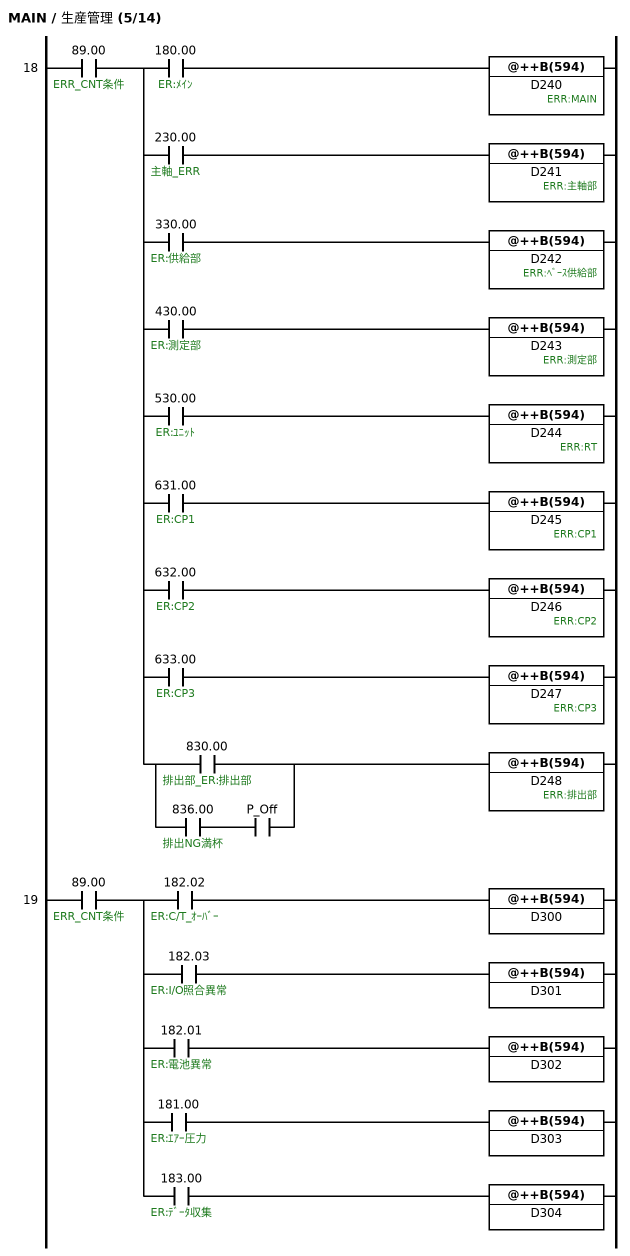
; [picture p24: MAIN / 生産管理, rungs 18-19]
; rung 18
LD 89.00  ; ERR_CNT条件
OUT TR0
AND 180.00  ; ER:ﾒｲﾝ
@++B(594) D240  ; ERR:MAIN
LD TR0
AND 230.00  ; 主軸_ERR
@++B(594) D241  ; ERR:主軸部
LD TR0
AND 330.00  ; ER:供給部
@++B(594) D242  ; ERR:ﾍﾞｰｽ供給部
LD TR0
AND 430.00  ; ER:測定部
@++B(594) D243  ; ERR:測定部
LD TR0
AND 530.00  ; ER:ﾕﾆｯﾄ
@++B(594) D244  ; ERR:RT
LD TR0
AND 631.00  ; ER:CP1
@++B(594) D245  ; ERR:CP1
LD TR0
AND 632.00  ; ER:CP2
@++B(594) D246  ; ERR:CP2
LD TR0
AND 633.00  ; ER:CP3
@++B(594) D247  ; ERR:CP3
LD TR0
LD 830.00  ; 排出部_ER:排出部
LD 836.00  ; 排出NG満杯
AND P_Off
ORLD
ANDLD
@++B(594) D248  ; ERR:排出部
; rung 19
LD 89.00  ; ERR_CNT条件
OUT TR0
AND 182.02  ; ER:C/T_ｵｰﾊﾞｰ
@++B(594) D300
LD TR0
AND 182.03  ; ER:I/O照合異常
@++B(594) D301
LD TR0
AND 182.01  ; ER:電池異常
@++B(594) D302
LD TR0
AND 181.00  ; ER:ｴｱｰ圧力
@++B(594) D303
LD TR0
AND 183.00  ; ER:ﾃﾞｰﾀ収集
@++B(594) D304

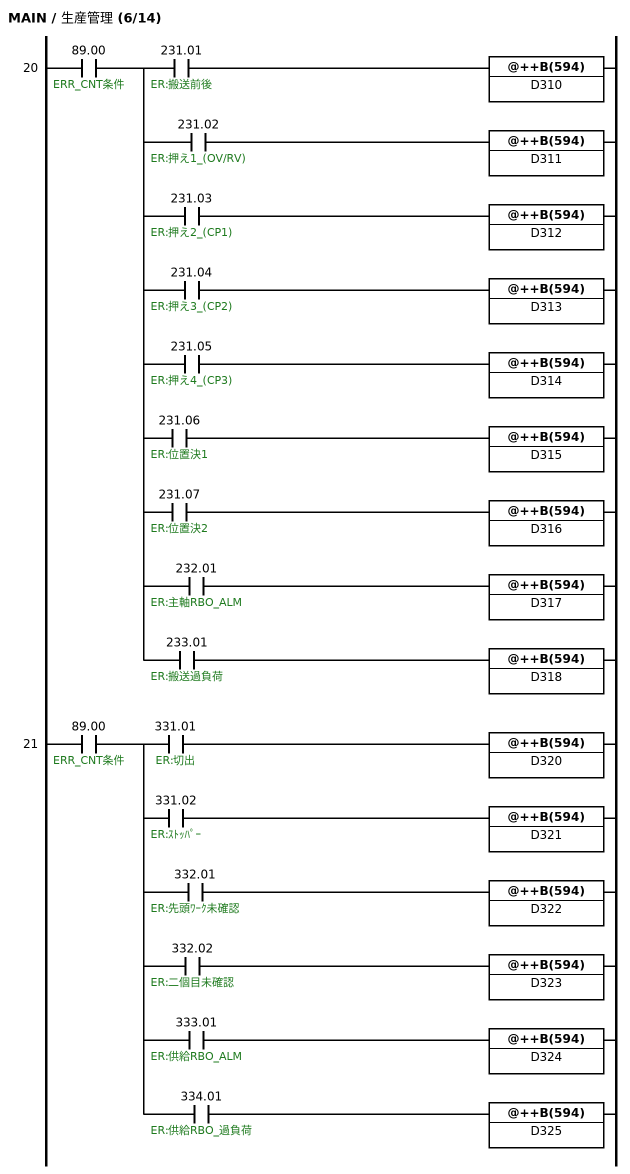
; rung 20
LD 89.00  ; ERR_CNT条件
OUT TR0
AND 231.01  ; ER:搬送前後
@++B(594) D310
LD TR0
AND 231.02  ; ER:押え1_(OV/RV)
@++B(594) D311
LD TR0
AND 231.03  ; ER:押え2_(CP1)
@++B(594) D312
LD TR0
AND 231.04  ; ER:押え3_(CP2)
@++B(594) D313
LD TR0
AND 231.05  ; ER:押え4_(CP3)
@++B(594) D314
LD TR0
AND 231.06  ; ER:位置決1
@++B(594) D315
LD TR0
AND 231.07  ; ER:位置決2
@++B(594) D316
LD TR0
AND 232.01  ; ER:主軸RBO_ALM
@++B(594) D317
LD TR0
AND 233.01  ; ER:搬送過負荷
@++B(594) D318
; rung 21
LD 89.00  ; ERR_CNT条件
OUT TR0
AND 331.01  ; ER:切出
@++B(594) D320
LD TR0
AND 331.02  ; ER:ｽﾄｯﾊﾟｰ
@++B(594) D321
LD TR0
AND 332.01  ; ER:先頭ﾜｰｸ未確認
@++B(594) D322
LD TR0
AND 332.02  ; ER:二個目未確認
@++B(594) D323
LD TR0
AND 333.01  ; ER:供給RBO_ALM
@++B(594) D324
LD TR0
AND 334.01  ; ER:供給RBO_過負荷
@++B(594) D325

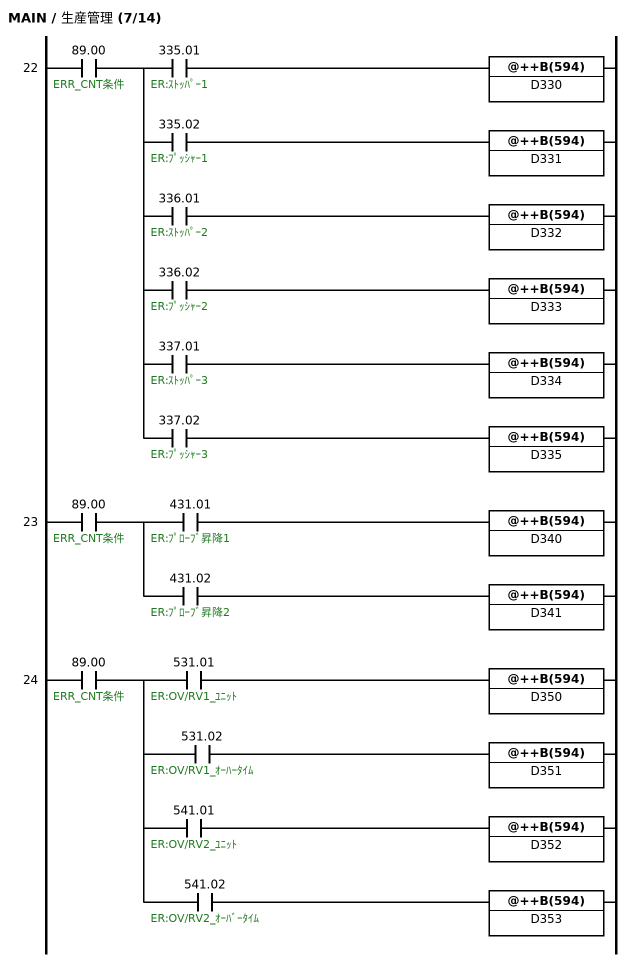
; rung 22
LD 89.00  ; ERR_CNT条件
OUT TR0
AND 335.01  ; ER:ｽﾄｯﾊﾟｰ1
@++B(594) D330
LD TR0
AND 335.02  ; ER:ﾌﾟｯｼｬｰ1
@++B(594) D331
LD TR0
AND 336.01  ; ER:ｽﾄｯﾊﾟｰ2
@++B(594) D332
LD TR0
AND 336.02  ; ER:ﾌﾟｯｼｬｰ2
@++B(594) D333
LD TR0
AND 337.01  ; ER:ｽﾄｯﾊﾟｰ3
@++B(594) D334
LD TR0
AND 337.02  ; ER:ﾌﾟｯｼｬｰ3
@++B(594) D335
; rung 23
LD 89.00  ; ERR_CNT条件
OUT TR0
AND 431.01  ; ER:ﾌﾟﾛｰﾌﾞ昇降1
@++B(594) D340
LD TR0
AND 431.02  ; ER:ﾌﾟﾛｰﾌﾞ昇降2
@++B(594) D341
; rung 24
LD 89.00  ; ERR_CNT条件
OUT TR0
AND 531.01  ; ER:OV/RV1_ﾕﾆｯﾄ
@++B(594) D350
LD TR0
AND 531.02  ; ER:OV/RV1_ｵｰﾊｰﾀｲﾑ
@++B(594) D351
LD TR0
AND 541.01  ; ER:OV/RV2_ﾕﾆｯﾄ
@++B(594) D352
LD TR0
AND 541.02  ; ER:OV/RV2_ｵｰﾊﾞｰﾀｲﾑ
@++B(594) D353

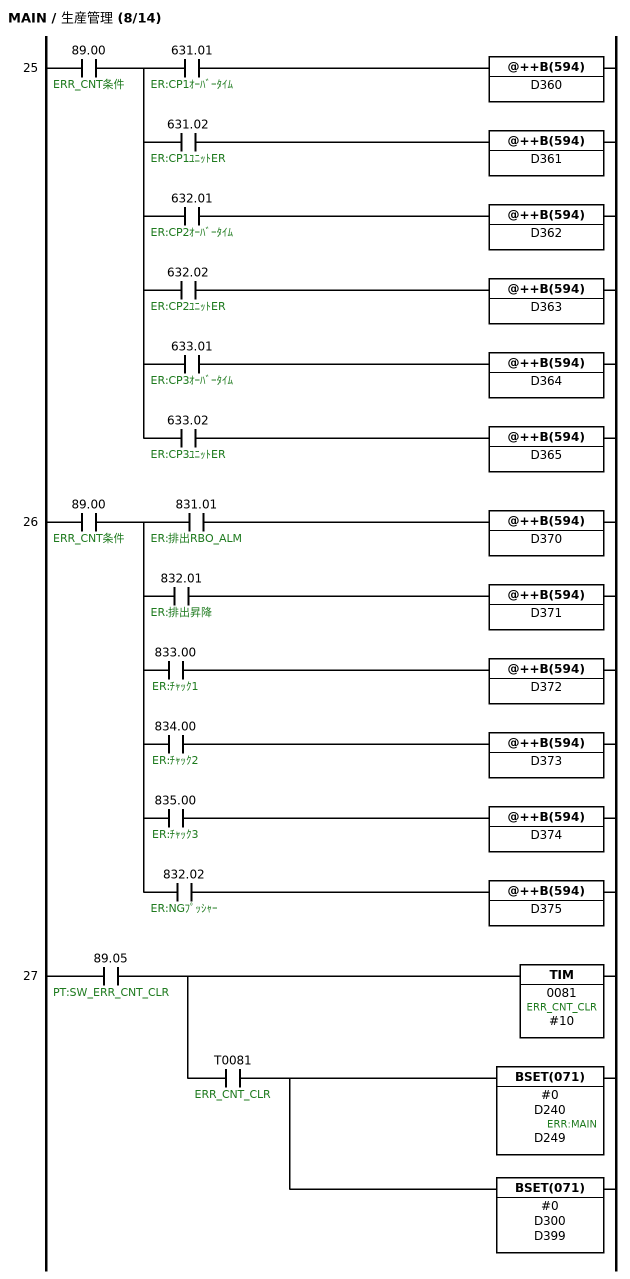
; rung 25
LD 89.00  ; ERR_CNT条件
OUT TR0
AND 631.01  ; ER:CP1ｵｰﾊﾞｰﾀｲﾑ
@++B(594) D360
LD TR0
AND 631.02  ; ER:CP1ﾕﾆｯﾄER
@++B(594) D361
LD TR0
AND 632.01  ; ER:CP2ｵｰﾊﾞｰﾀｲﾑ
@++B(594) D362
LD TR0
AND 632.02  ; ER:CP2ﾕﾆｯﾄER
@++B(594) D363
LD TR0
AND 633.01  ; ER:CP3ｵｰﾊﾞｰﾀｲﾑ
@++B(594) D364
LD TR0
AND 633.02  ; ER:CP3ﾕﾆｯﾄER
@++B(594) D365
; rung 26
LD 89.00  ; ERR_CNT条件
OUT TR0
AND 831.01  ; ER:排出RBO_ALM
@++B(594) D370
LD TR0
AND 832.01  ; ER:排出昇降
@++B(594) D371
LD TR0
AND 833.00  ; ER:ﾁｬｯｸ1
@++B(594) D372
LD TR0
AND 834.00  ; ER:ﾁｬｯｸ2
@++B(594) D373
LD TR0
AND 835.00  ; ER:ﾁｬｯｸ3
@++B(594) D374
LD TR0
AND 832.02  ; ER:NGﾌﾟｯｼｬｰ
@++B(594) D375
; rung 27
LD 89.05  ; PT:SW_ERR_CNT_CLR
TIM 0081 #10  ; ERR_CNT_CLR
AND T0081  ; ERR_CNT_CLR
BSET(071) #0 D240 D249  ; ERR:MAIN
BSET(071) #0 D300 D399

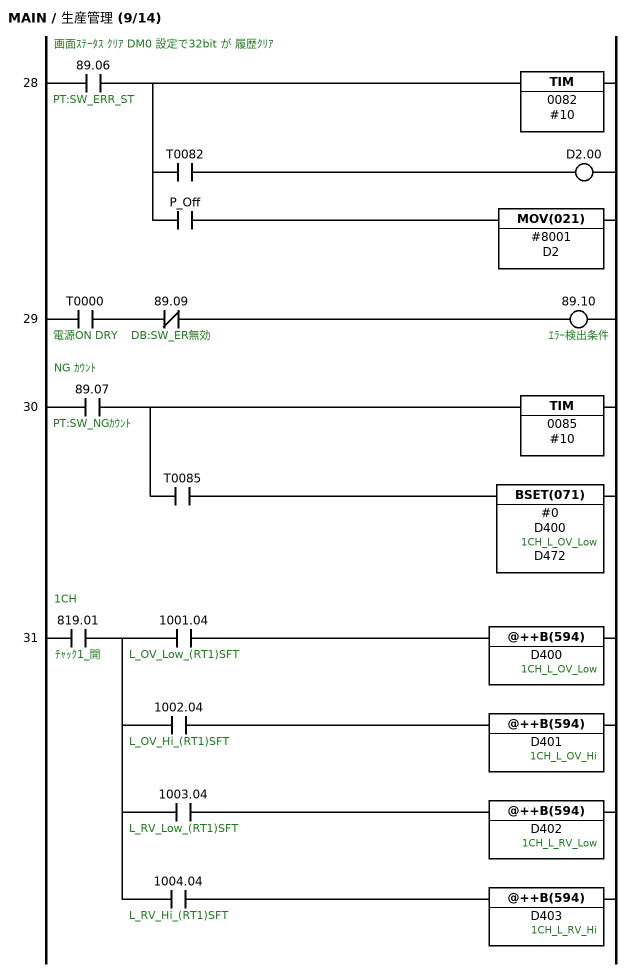
; rung 28: 画面ｽﾃｰﾀｽ ｸﾘｱ DM0 設定で32bit が 履歴ｸﾘｱ
LD 89.06  ; PT:SW_ERR_ST
OUT TR0
TIM 0082 #10
AND T0082
OUT D2.00
LD TR0
AND P_Off
MOV(021) #8001 D2
; rung 29
LD T0000  ; 電源ON DRY
ANDNOT 89.09  ; DB:SW_ER無効
OUT 89.10  ; ｴﾗｰ検出条件
; rung 30: NG ｶｳﾝﾄ
LD 89.07  ; PT:SW_NGｶｳﾝﾄ
TIM 0085 #10
AND T0085
BSET(071) #0 D400 D472  ; 1CH_L_OV_Low
; rung 31: 1CH
LD 819.01  ; ﾁｬｯｸ1_開
OUT TR0
AND 1001.04  ; L_OV_Low_(RT1)SFT
@++B(594) D400  ; 1CH_L_OV_Low
LD TR0
AND 1002.04  ; L_OV_Hi_(RT1)SFT
@++B(594) D401  ; 1CH_L_OV_Hi
LD TR0
AND 1003.04  ; L_RV_Low_(RT1)SFT
@++B(594) D402  ; 1CH_L_RV_Low
LD TR0
AND 1004.04  ; L_RV_Hi_(RT1)SFT
@++B(594) D403  ; 1CH_L_RV_Hi

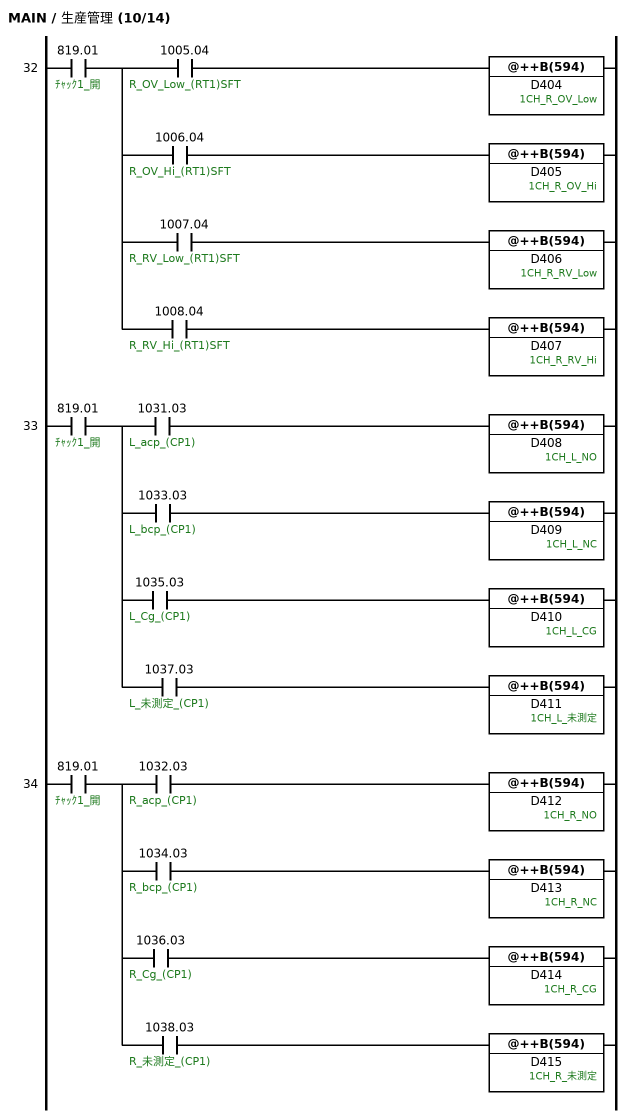
; rung 32
LD 819.01  ; ﾁｬｯｸ1_開
OUT TR0
AND 1005.04  ; R_OV_Low_(RT1)SFT
@++B(594) D404  ; 1CH_R_OV_Low
LD TR0
AND 1006.04  ; R_OV_Hi_(RT1)SFT
@++B(594) D405  ; 1CH_R_OV_Hi
LD TR0
AND 1007.04  ; R_RV_Low_(RT1)SFT
@++B(594) D406  ; 1CH_R_RV_Low
LD TR0
AND 1008.04  ; R_RV_Hi_(RT1)SFT
@++B(594) D407  ; 1CH_R_RV_Hi
; rung 33
LD 819.01  ; ﾁｬｯｸ1_開
OUT TR0
AND 1031.03  ; L_acp_(CP1)
@++B(594) D408  ; 1CH_L_NO
LD TR0
AND 1033.03  ; L_bcp_(CP1)
@++B(594) D409  ; 1CH_L_NC
LD TR0
AND 1035.03  ; L_Cg_(CP1)
@++B(594) D410  ; 1CH_L_CG
LD TR0
AND 1037.03  ; L_未測定_(CP1)
@++B(594) D411  ; 1CH_L_未測定
; rung 34
LD 819.01  ; ﾁｬｯｸ1_開
OUT TR0
AND 1032.03  ; R_acp_(CP1)
@++B(594) D412  ; 1CH_R_NO
LD TR0
AND 1034.03  ; R_bcp_(CP1)
@++B(594) D413  ; 1CH_R_NC
LD TR0
AND 1036.03  ; R_Cg_(CP1)
@++B(594) D414  ; 1CH_R_CG
LD TR0
AND 1038.03  ; R_未測定_(CP1)
@++B(594) D415  ; 1CH_R_未測定

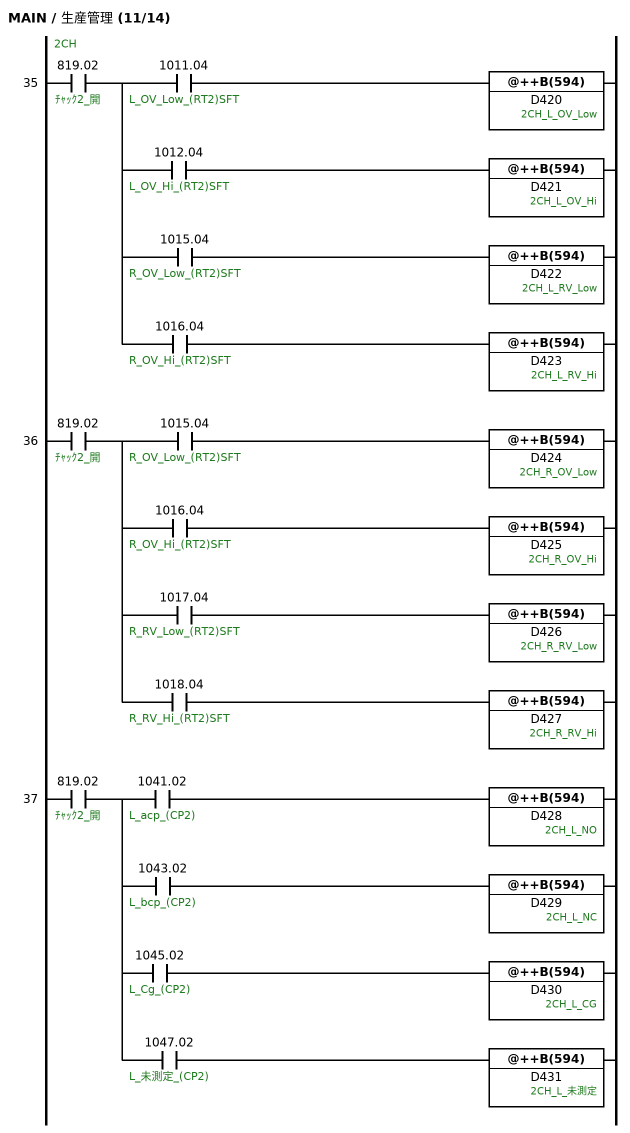
; rung 35: 2CH
LD 819.02  ; ﾁｬｯｸ2_開
OUT TR0
AND 1011.04  ; L_OV_Low_(RT2)SFT
@++B(594) D420  ; 2CH_L_OV_Low
LD TR0
AND 1012.04  ; L_OV_Hi_(RT2)SFT
@++B(594) D421  ; 2CH_L_OV_Hi
LD TR0
AND 1015.04  ; R_OV_Low_(RT2)SFT
@++B(594) D422  ; 2CH_L_RV_Low
LD TR0
AND 1016.04  ; R_OV_Hi_(RT2)SFT
@++B(594) D423  ; 2CH_L_RV_Hi
; rung 36
LD 819.02  ; ﾁｬｯｸ2_開
OUT TR0
AND 1015.04  ; R_OV_Low_(RT2)SFT
@++B(594) D424  ; 2CH_R_OV_Low
LD TR0
AND 1016.04  ; R_OV_Hi_(RT2)SFT
@++B(594) D425  ; 2CH_R_OV_Hi
LD TR0
AND 1017.04  ; R_RV_Low_(RT2)SFT
@++B(594) D426  ; 2CH_R_RV_Low
LD TR0
AND 1018.04  ; R_RV_Hi_(RT2)SFT
@++B(594) D427  ; 2CH_R_RV_Hi
; rung 37
LD 819.02  ; ﾁｬｯｸ2_開
OUT TR0
AND 1041.02  ; L_acp_(CP2)
@++B(594) D428  ; 2CH_L_NO
LD TR0
AND 1043.02  ; L_bcp_(CP2)
@++B(594) D429  ; 2CH_L_NC
LD TR0
AND 1045.02  ; L_Cg_(CP2)
@++B(594) D430  ; 2CH_L_CG
LD TR0
AND 1047.02  ; L_未測定_(CP2)
@++B(594) D431  ; 2CH_L_未測定

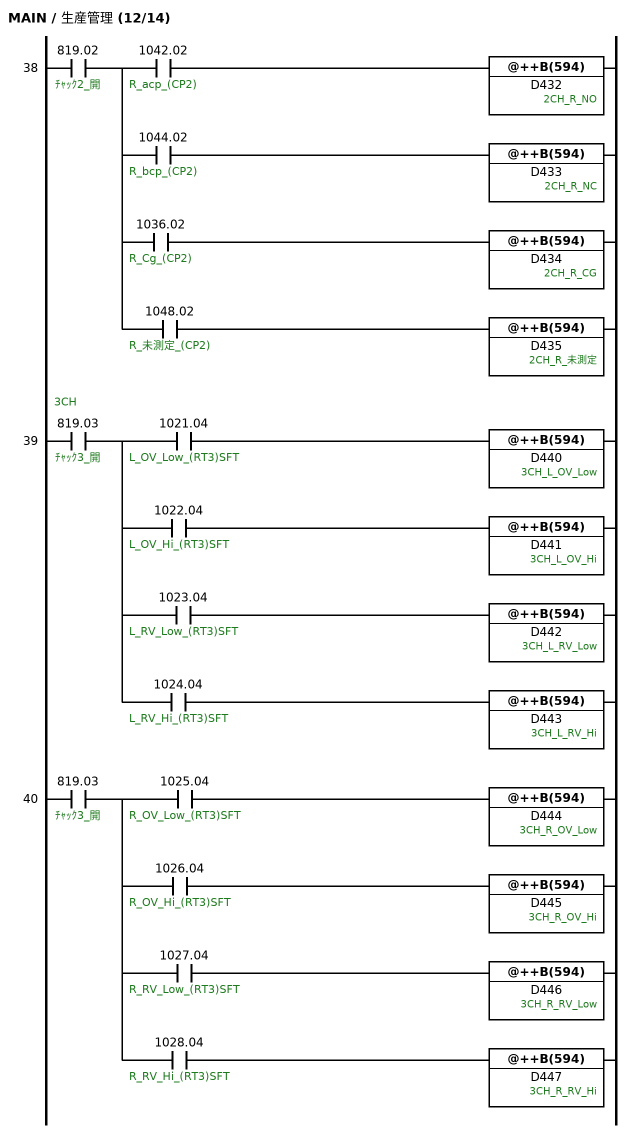
; rung 38
LD 819.02  ; ﾁｬｯｸ2_開
OUT TR0
AND 1042.02  ; R_acp_(CP2)
@++B(594) D432  ; 2CH_R_NO
LD TR0
AND 1044.02  ; R_bcp_(CP2)
@++B(594) D433  ; 2CH_R_NC
LD TR0
AND 1036.02  ; R_Cg_(CP2)
@++B(594) D434  ; 2CH_R_CG
LD TR0
AND 1048.02  ; R_未測定_(CP2)
@++B(594) D435  ; 2CH_R_未測定
; rung 39: 3CH
LD 819.03  ; ﾁｬｯｸ3_開
OUT TR0
AND 1021.04  ; L_OV_Low_(RT3)SFT
@++B(594) D440  ; 3CH_L_OV_Low
LD TR0
AND 1022.04  ; L_OV_Hi_(RT3)SFT
@++B(594) D441  ; 3CH_L_OV_Hi
LD TR0
AND 1023.04  ; L_RV_Low_(RT3)SFT
@++B(594) D442  ; 3CH_L_RV_Low
LD TR0
AND 1024.04  ; L_RV_Hi_(RT3)SFT
@++B(594) D443  ; 3CH_L_RV_Hi
; rung 40
LD 819.03  ; ﾁｬｯｸ3_開
OUT TR0
AND 1025.04  ; R_OV_Low_(RT3)SFT
@++B(594) D444  ; 3CH_R_OV_Low
LD TR0
AND 1026.04  ; R_OV_Hi_(RT3)SFT
@++B(594) D445  ; 3CH_R_OV_Hi
LD TR0
AND 1027.04  ; R_RV_Low_(RT3)SFT
@++B(594) D446  ; 3CH_R_RV_Low
LD TR0
AND 1028.04  ; R_RV_Hi_(RT3)SFT
@++B(594) D447  ; 3CH_R_RV_Hi

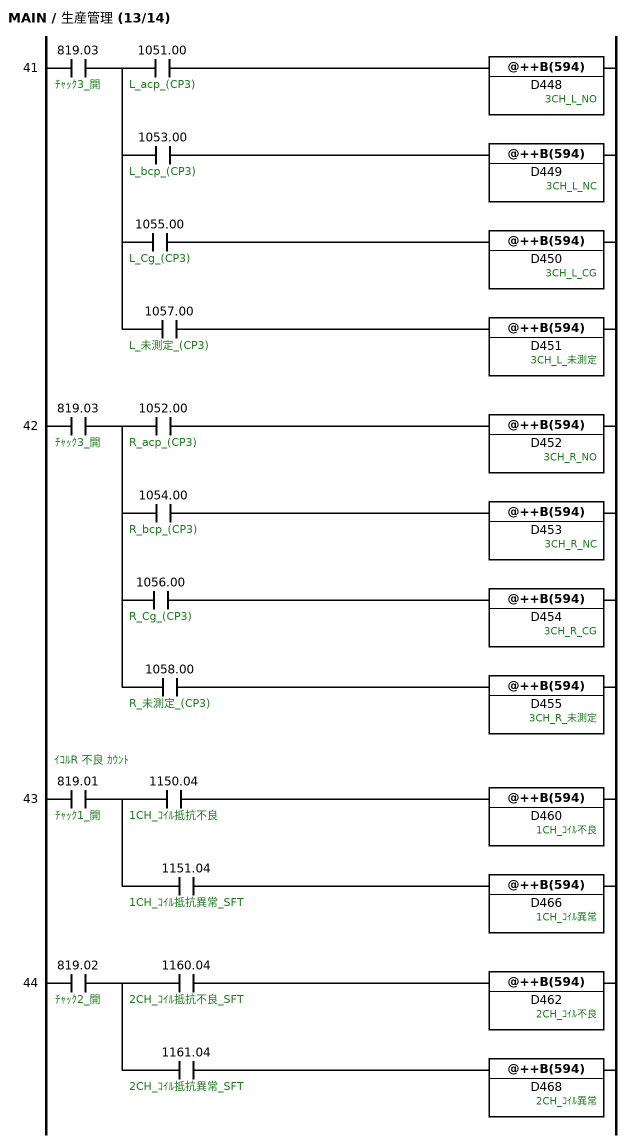
; rung 41
LD 819.03  ; ﾁｬｯｸ3_開
OUT TR0
AND 1051.00  ; L_acp_(CP3)
@++B(594) D448  ; 3CH_L_NO
LD TR0
AND 1053.00  ; L_bcp_(CP3)
@++B(594) D449  ; 3CH_L_NC
LD TR0
AND 1055.00  ; L_Cg_(CP3)
@++B(594) D450  ; 3CH_L_CG
LD TR0
AND 1057.00  ; L_未測定_(CP3)
@++B(594) D451  ; 3CH_L_未測定
; rung 42
LD 819.03  ; ﾁｬｯｸ3_開
OUT TR0
AND 1052.00  ; R_acp_(CP3)
@++B(594) D452  ; 3CH_R_NO
LD TR0
AND 1054.00  ; R_bcp_(CP3)
@++B(594) D453  ; 3CH_R_NC
LD TR0
AND 1056.00  ; R_Cg_(CP3)
@++B(594) D454  ; 3CH_R_CG
LD TR0
AND 1058.00  ; R_未測定_(CP3)
@++B(594) D455  ; 3CH_R_未測定
; rung 43: ｲｺﾙR 不良 ｶｳﾝﾄ
LD 819.01  ; ﾁｬｯｸ1_開
OUT TR0
AND 1150.04  ; 1CH_ｺｲﾙ抵抗不良
@++B(594) D460  ; 1CH_ｺｲﾙ不良
LD TR0
AND 1151.04  ; 1CH_ｺｲﾙ抵抗異常_SFT
@++B(594) D466  ; 1CH_ｺｲﾙ異常
; rung 44
LD 819.02  ; ﾁｬｯｸ2_開
OUT TR0
AND 1160.04  ; 2CH_ｺｲﾙ抵抗不良_SFT
@++B(594) D462  ; 2CH_ｺｲﾙ不良
LD TR0
AND 1161.04  ; 2CH_ｺｲﾙ抵抗異常_SFT
@++B(594) D468  ; 2CH_ｺｲﾙ異常

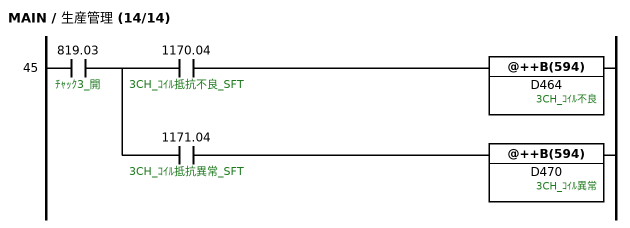
; rung 45
LD 819.03  ; ﾁｬｯｸ3_開
OUT TR0
AND 1170.04  ; 3CH_ｺｲﾙ抵抗不良_SFT
@++B(594) D464  ; 3CH_ｺｲﾙ不良
LD TR0
AND 1171.04  ; 3CH_ｺｲﾙ抵抗異常_SFT
@++B(594) D470  ; 3CH_ｺｲﾙ異常

### Section ERR

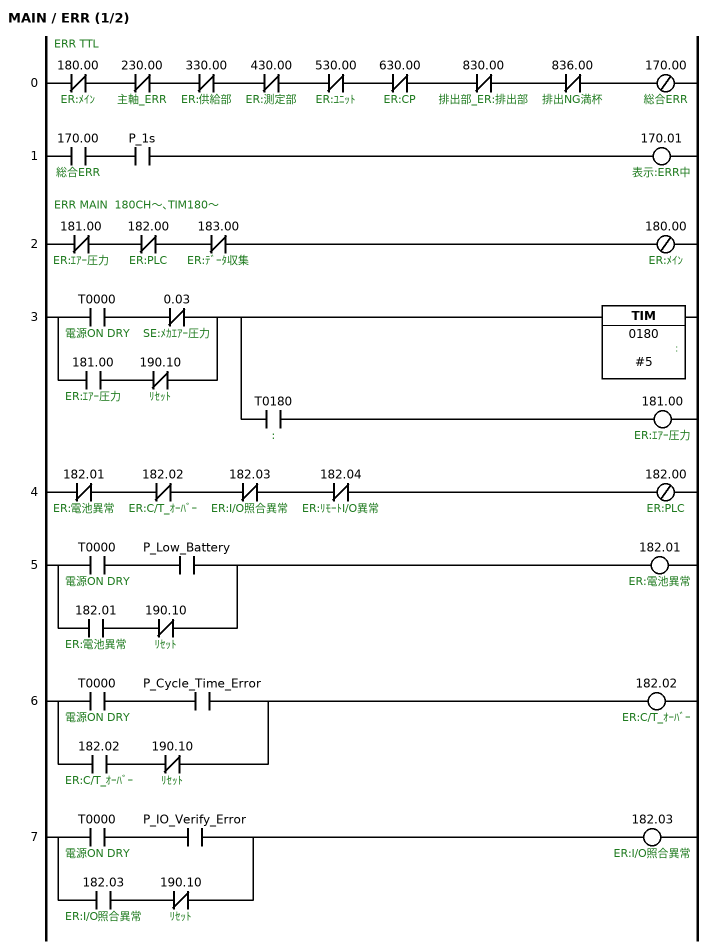
; rung 0: ERR TTL
LDNOT 180.00  ; ER:ﾒｲﾝ
ANDNOT 230.00  ; 主軸_ERR
ANDNOT 330.00  ; ER:供給部
ANDNOT 430.00  ; ER:測定部
ANDNOT 530.00  ; ER:ﾕﾆｯﾄ
ANDNOT 630.00  ; ER:CP
ANDNOT 830.00  ; 排出部_ER:排出部
ANDNOT 836.00  ; 排出NG満杯
OUTNOT 170.00  ; 総合ERR
; rung 1
LD 170.00  ; 総合ERR
AND P_1s
OUT 170.01  ; 表示:ERR中
; rung 2: ERR MAIN  180CH～､TIM180～
LDNOT 181.00  ; ER:ｴｱｰ圧力
ANDNOT 182.00  ; ER:PLC
ANDNOT 183.00  ; ER:ﾃﾞｰﾀ収集
OUTNOT 180.00  ; ER:ﾒｲﾝ
; rung 3
LD T0000  ; 電源ON DRY
ANDNOT 0.03  ; SE:ﾒｶｴｱｰ圧力
LD 181.00  ; ER:ｴｱｰ圧力
ANDNOT 190.10  ; ﾘｾｯﾄ
ORLD
TIM 0180 #5  ; :
AND T0180  ; :
OUT 181.00  ; ER:ｴｱｰ圧力
; rung 4
LDNOT 182.01  ; ER:電池異常
ANDNOT 182.02  ; ER:C/T_ｵｰﾊﾞｰ
ANDNOT 182.03  ; ER:I/O照合異常
ANDNOT 182.04  ; ER:ﾘﾓｰﾄI/O異常
OUTNOT 182.00  ; ER:PLC
; rung 5
LD T0000  ; 電源ON DRY
AND P_Low_Battery
LD 182.01  ; ER:電池異常
ANDNOT 190.10  ; ﾘｾｯﾄ
ORLD
OUT 182.01  ; ER:電池異常
; rung 6
LD T0000  ; 電源ON DRY
AND P_Cycle_Time_Error
LD 182.02  ; ER:C/T_ｵｰﾊﾞｰ
ANDNOT 190.10  ; ﾘｾｯﾄ
ORLD
OUT 182.02  ; ER:C/T_ｵｰﾊﾞｰ
; rung 7
LD T0000  ; 電源ON DRY
AND P_IO_Verify_Error
LD 182.03  ; ER:I/O照合異常
ANDNOT 190.10  ; ﾘｾｯﾄ
ORLD
OUT 182.03  ; ER:I/O照合異常

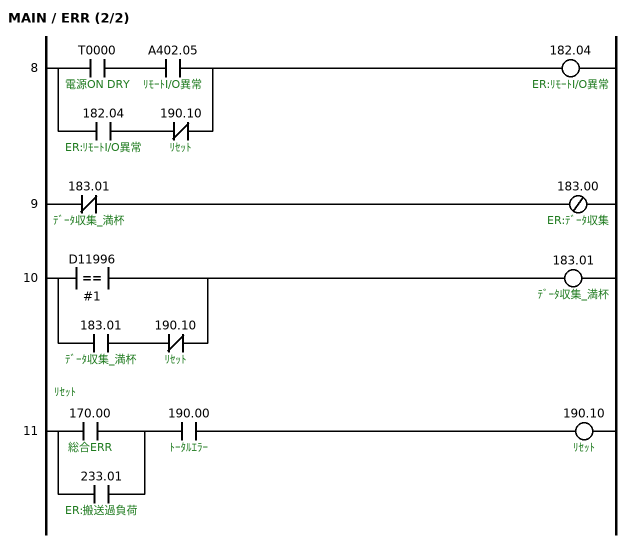
; rung 8
LD T0000  ; 電源ON DRY
AND A402.05  ; ﾘﾓｰﾄI/O異常
LD 182.04  ; ER:ﾘﾓｰﾄI/O異常
ANDNOT 190.10  ; ﾘｾｯﾄ
ORLD
OUT 182.04  ; ER:ﾘﾓｰﾄI/O異常
; rung 9
LDNOT 183.01  ; ﾃﾞｰﾀ収集_満杯
OUTNOT 183.00  ; ER:ﾃﾞｰﾀ収集
; rung 10
LD=(300) D11996 #1
LD 183.01  ; ﾃﾞｰﾀ収集_満杯
ANDNOT 190.10  ; ﾘｾｯﾄ
ORLD
OUT 183.01  ; ﾃﾞｰﾀ収集_満杯
; rung 11: ﾘｾｯﾄ
LD 170.00  ; 総合ERR
OR 233.01  ; ER:搬送過負荷
AND 190.00  ; ﾄｰﾀﾙｴﾗｰ
OUT 190.10  ; ﾘｾｯﾄ

### Section 手動操作

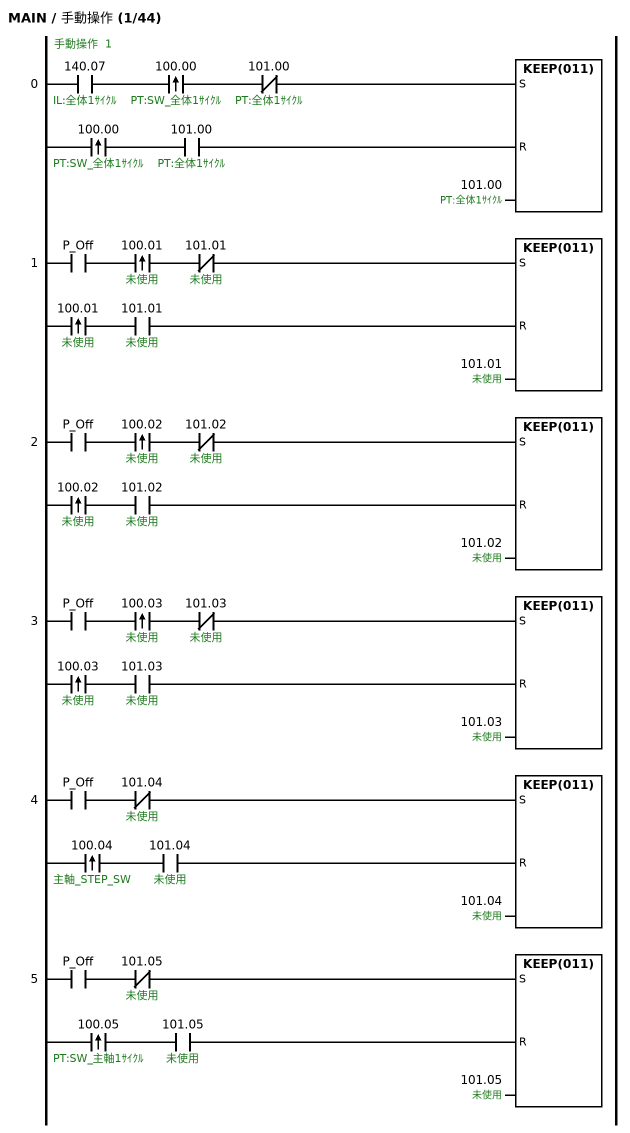
; rung 0: 手動操作  1
LD 140.07  ; IL:全体1ｻｲｸﾙ
@AND 100.00  ; PT:SW_全体1ｻｲｸﾙ
ANDNOT 101.00  ; PT:全体1ｻｲｸﾙ
@LD 100.00  ; PT:SW_全体1ｻｲｸﾙ
AND 101.00  ; PT:全体1ｻｲｸﾙ
KEEP(011) 101.00  ; PT:全体1ｻｲｸﾙ
; rung 1
LD P_Off
@AND 100.01  ; 未使用
ANDNOT 101.01  ; 未使用
@LD 100.01  ; 未使用
AND 101.01  ; 未使用
KEEP(011) 101.01  ; 未使用
; rung 2
LD P_Off
@AND 100.02  ; 未使用
ANDNOT 101.02  ; 未使用
@LD 100.02  ; 未使用
AND 101.02  ; 未使用
KEEP(011) 101.02  ; 未使用
; rung 3
LD P_Off
@AND 100.03  ; 未使用
ANDNOT 101.03  ; 未使用
@LD 100.03  ; 未使用
AND 101.03  ; 未使用
KEEP(011) 101.03  ; 未使用
; rung 4
LD P_Off
ANDNOT 101.04  ; 未使用
@LD 100.04  ; 主軸_STEP_SW
AND 101.04  ; 未使用
KEEP(011) 101.04  ; 未使用
; rung 5
LD P_Off
ANDNOT 101.05  ; 未使用
@LD 100.05  ; PT:SW_主軸1ｻｲｸﾙ
AND 101.05  ; 未使用
KEEP(011) 101.05  ; 未使用

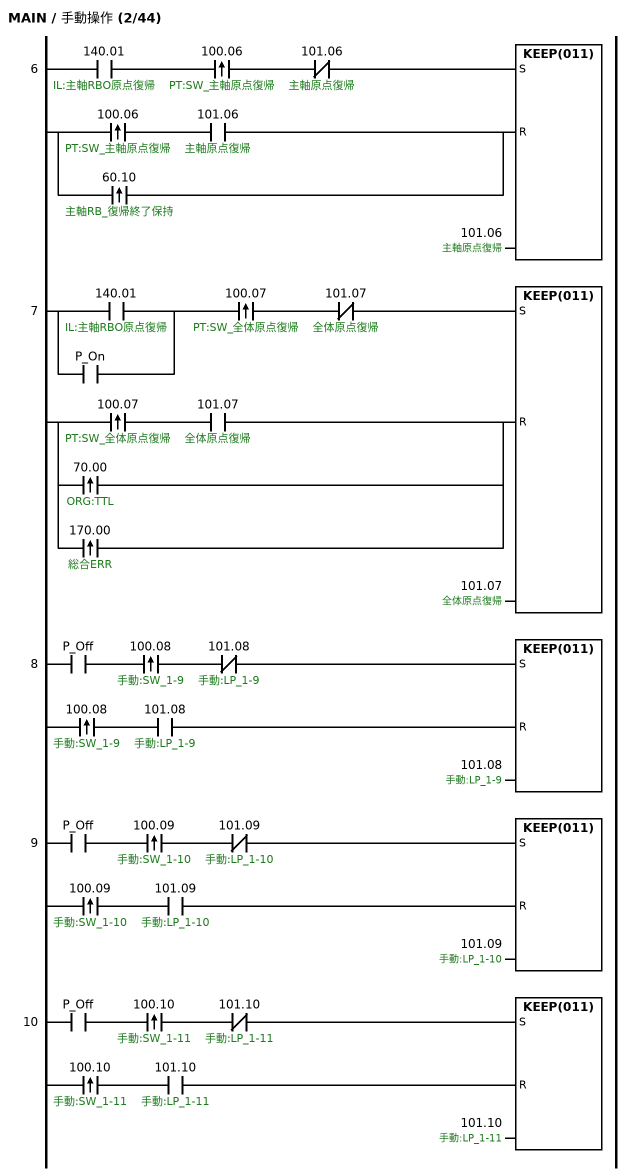
; rung 6
LD 140.01  ; IL:主軸RBO原点復帰
@AND 100.06  ; PT:SW_主軸原点復帰
ANDNOT 101.06  ; 主軸原点復帰
@LD 100.06  ; PT:SW_主軸原点復帰
AND 101.06  ; 主軸原点復帰
@OR 60.10  ; 主軸RB_復帰終了保持
KEEP(011) 101.06  ; 主軸原点復帰
; rung 7
LD 140.01  ; IL:主軸RBO原点復帰
OR P_On
@AND 100.07  ; PT:SW_全体原点復帰
ANDNOT 101.07  ; 全体原点復帰
@LD 100.07  ; PT:SW_全体原点復帰
AND 101.07  ; 全体原点復帰
@OR 70.00  ; ORG:TTL
@OR 170.00  ; 総合ERR
KEEP(011) 101.07  ; 全体原点復帰
; rung 8
LD P_Off
@AND 100.08  ; 手動:SW_1-9
ANDNOT 101.08  ; 手動:LP_1-9
@LD 100.08  ; 手動:SW_1-9
AND 101.08  ; 手動:LP_1-9
KEEP(011) 101.08  ; 手動:LP_1-9
; rung 9
LD P_Off
@AND 100.09  ; 手動:SW_1-10
ANDNOT 101.09  ; 手動:LP_1-10
@LD 100.09  ; 手動:SW_1-10
AND 101.09  ; 手動:LP_1-10
KEEP(011) 101.09  ; 手動:LP_1-10
; rung 10
LD P_Off
@AND 100.10  ; 手動:SW_1-11
ANDNOT 101.10  ; 手動:LP_1-11
@LD 100.10  ; 手動:SW_1-11
AND 101.10  ; 手動:LP_1-11
KEEP(011) 101.10  ; 手動:LP_1-11

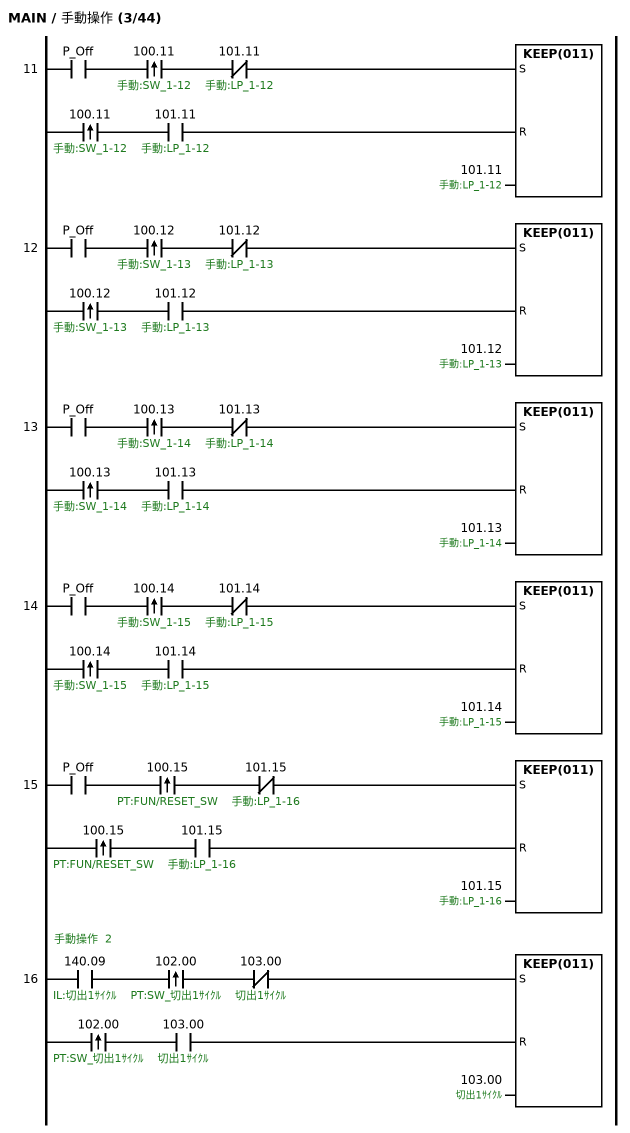
; rung 11
LD P_Off
@AND 100.11  ; 手動:SW_1-12
ANDNOT 101.11  ; 手動:LP_1-12
@LD 100.11  ; 手動:SW_1-12
AND 101.11  ; 手動:LP_1-12
KEEP(011) 101.11  ; 手動:LP_1-12
; rung 12
LD P_Off
@AND 100.12  ; 手動:SW_1-13
ANDNOT 101.12  ; 手動:LP_1-13
@LD 100.12  ; 手動:SW_1-13
AND 101.12  ; 手動:LP_1-13
KEEP(011) 101.12  ; 手動:LP_1-13
; rung 13
LD P_Off
@AND 100.13  ; 手動:SW_1-14
ANDNOT 101.13  ; 手動:LP_1-14
@LD 100.13  ; 手動:SW_1-14
AND 101.13  ; 手動:LP_1-14
KEEP(011) 101.13  ; 手動:LP_1-14
; rung 14
LD P_Off
@AND 100.14  ; 手動:SW_1-15
ANDNOT 101.14  ; 手動:LP_1-15
@LD 100.14  ; 手動:SW_1-15
AND 101.14  ; 手動:LP_1-15
KEEP(011) 101.14  ; 手動:LP_1-15
; rung 15
LD P_Off
@AND 100.15  ; PT:FUN/RESET_SW
ANDNOT 101.15  ; 手動:LP_1-16
@LD 100.15  ; PT:FUN/RESET_SW
AND 101.15  ; 手動:LP_1-16
KEEP(011) 101.15  ; 手動:LP_1-16
; rung 16: 手動操作  2
LD 140.09  ; IL:切出1ｻｲｸﾙ
@AND 102.00  ; PT:SW_切出1ｻｲｸﾙ
ANDNOT 103.00  ; 切出1ｻｲｸﾙ
@LD 102.00  ; PT:SW_切出1ｻｲｸﾙ
AND 103.00  ; 切出1ｻｲｸﾙ
KEEP(011) 103.00  ; 切出1ｻｲｸﾙ

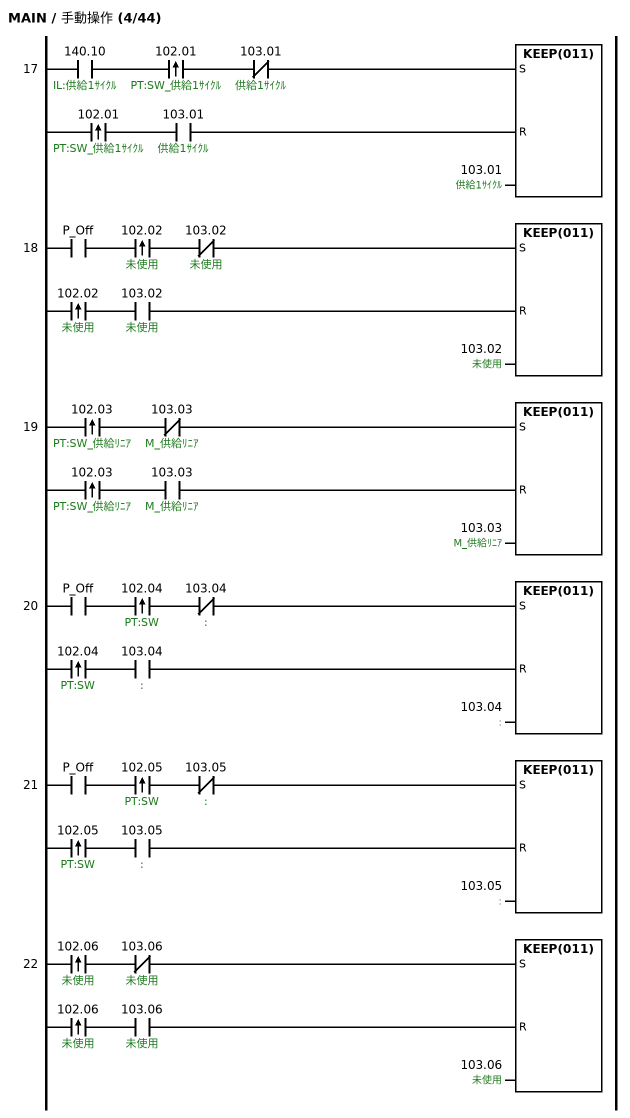
; rung 17
LD 140.10  ; IL:供給1ｻｲｸﾙ
@AND 102.01  ; PT:SW_供給1ｻｲｸﾙ
ANDNOT 103.01  ; 供給1ｻｲｸﾙ
@LD 102.01  ; PT:SW_供給1ｻｲｸﾙ
AND 103.01  ; 供給1ｻｲｸﾙ
KEEP(011) 103.01  ; 供給1ｻｲｸﾙ
; rung 18
LD P_Off
@AND 102.02  ; 未使用
ANDNOT 103.02  ; 未使用
@LD 102.02  ; 未使用
AND 103.02  ; 未使用
KEEP(011) 103.02  ; 未使用
; rung 19
@LD 102.03  ; PT:SW_供給ﾘﾆｱ
ANDNOT 103.03  ; M_供給ﾘﾆｱ
@LD 102.03  ; PT:SW_供給ﾘﾆｱ
AND 103.03  ; M_供給ﾘﾆｱ
KEEP(011) 103.03  ; M_供給ﾘﾆｱ
; rung 20
LD P_Off
@AND 102.04  ; PT:SW
ANDNOT 103.04  ; :
@LD 102.04  ; PT:SW
AND 103.04  ; :
KEEP(011) 103.04  ; :
; rung 21
LD P_Off
@AND 102.05  ; PT:SW
ANDNOT 103.05  ; :
@LD 102.05  ; PT:SW
AND 103.05  ; :
KEEP(011) 103.05  ; :
; rung 22
@LD 102.06  ; 未使用
ANDNOT 103.06  ; 未使用
@LD 102.06  ; 未使用
AND 103.06  ; 未使用
KEEP(011) 103.06  ; 未使用

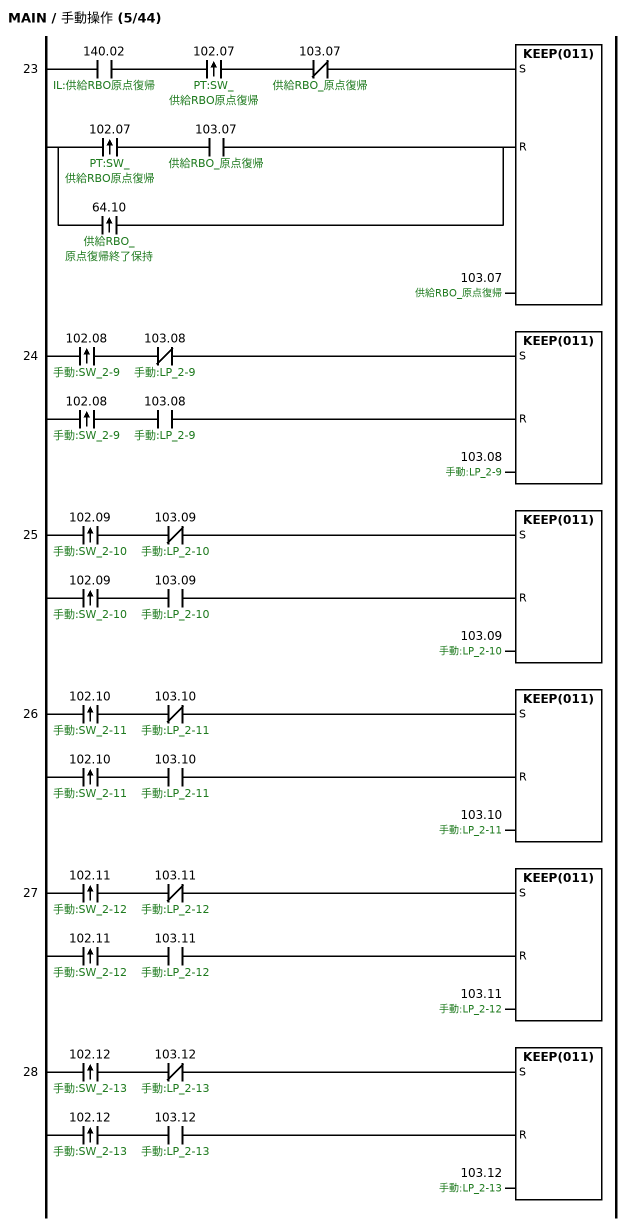
; rung 23
LD 140.02  ; IL:供給RBO原点復帰
@AND 102.07  ; PT:SW_供給RBO原点復帰
ANDNOT 103.07  ; 供給RBO_原点復帰
@LD 102.07  ; PT:SW_供給RBO原点復帰
AND 103.07  ; 供給RBO_原点復帰
@OR 64.10  ; 供給RBO_原点復帰終了保持
KEEP(011) 103.07  ; 供給RBO_原点復帰
; rung 24
@LD 102.08  ; 手動:SW_2-9
ANDNOT 103.08  ; 手動:LP_2-9
@LD 102.08  ; 手動:SW_2-9
AND 103.08  ; 手動:LP_2-9
KEEP(011) 103.08  ; 手動:LP_2-9
; rung 25
@LD 102.09  ; 手動:SW_2-10
ANDNOT 103.09  ; 手動:LP_2-10
@LD 102.09  ; 手動:SW_2-10
AND 103.09  ; 手動:LP_2-10
KEEP(011) 103.09  ; 手動:LP_2-10
; rung 26
@LD 102.10  ; 手動:SW_2-11
ANDNOT 103.10  ; 手動:LP_2-11
@LD 102.10  ; 手動:SW_2-11
AND 103.10  ; 手動:LP_2-11
KEEP(011) 103.10  ; 手動:LP_2-11
; rung 27
@LD 102.11  ; 手動:SW_2-12
ANDNOT 103.11  ; 手動:LP_2-12
@LD 102.11  ; 手動:SW_2-12
AND 103.11  ; 手動:LP_2-12
KEEP(011) 103.11  ; 手動:LP_2-12
; rung 28
@LD 102.12  ; 手動:SW_2-13
ANDNOT 103.12  ; 手動:LP_2-13
@LD 102.12  ; 手動:SW_2-13
AND 103.12  ; 手動:LP_2-13
KEEP(011) 103.12  ; 手動:LP_2-13

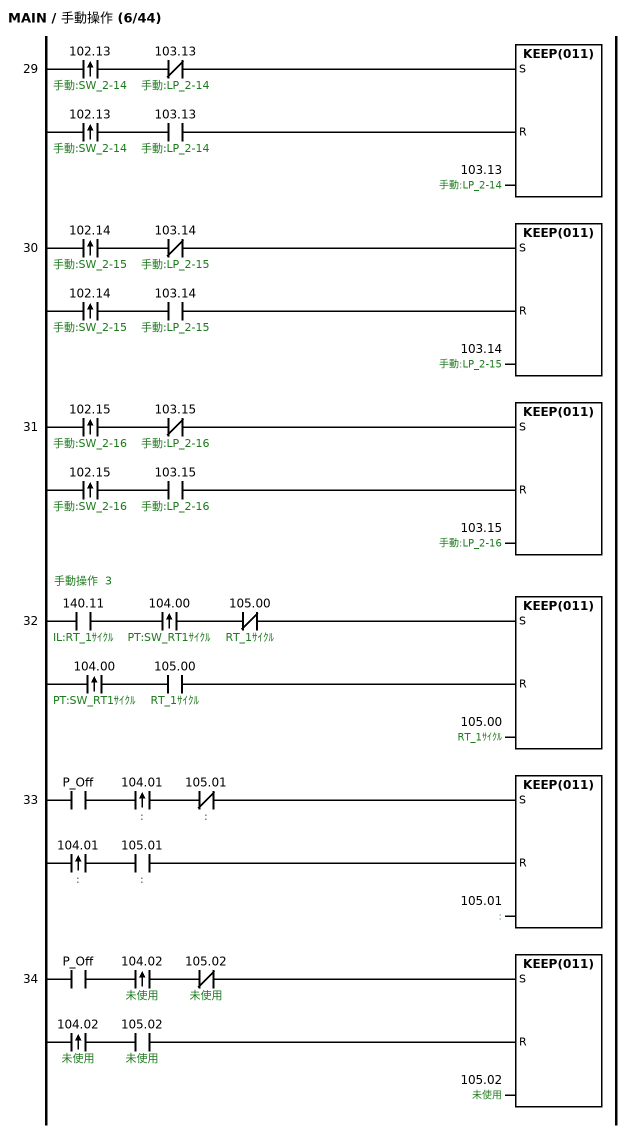
; rung 29
@LD 102.13  ; 手動:SW_2-14
ANDNOT 103.13  ; 手動:LP_2-14
@LD 102.13  ; 手動:SW_2-14
AND 103.13  ; 手動:LP_2-14
KEEP(011) 103.13  ; 手動:LP_2-14
; rung 30
@LD 102.14  ; 手動:SW_2-15
ANDNOT 103.14  ; 手動:LP_2-15
@LD 102.14  ; 手動:SW_2-15
AND 103.14  ; 手動:LP_2-15
KEEP(011) 103.14  ; 手動:LP_2-15
; rung 31
@LD 102.15  ; 手動:SW_2-16
ANDNOT 103.15  ; 手動:LP_2-16
@LD 102.15  ; 手動:SW_2-16
AND 103.15  ; 手動:LP_2-16
KEEP(011) 103.15  ; 手動:LP_2-16
; rung 32: 手動操作  3
LD 140.11  ; IL:RT_1ｻｲｸﾙ
@AND 104.00  ; PT:SW_RT1ｻｲｸﾙ
ANDNOT 105.00  ; RT_1ｻｲｸﾙ
@LD 104.00  ; PT:SW_RT1ｻｲｸﾙ
AND 105.00  ; RT_1ｻｲｸﾙ
KEEP(011) 105.00  ; RT_1ｻｲｸﾙ
; rung 33
LD P_Off
@AND 104.01  ; :
ANDNOT 105.01  ; :
@LD 104.01  ; :
AND 105.01  ; :
KEEP(011) 105.01  ; :
; rung 34
LD P_Off
@AND 104.02  ; 未使用
ANDNOT 105.02  ; 未使用
@LD 104.02  ; 未使用
AND 105.02  ; 未使用
KEEP(011) 105.02  ; 未使用

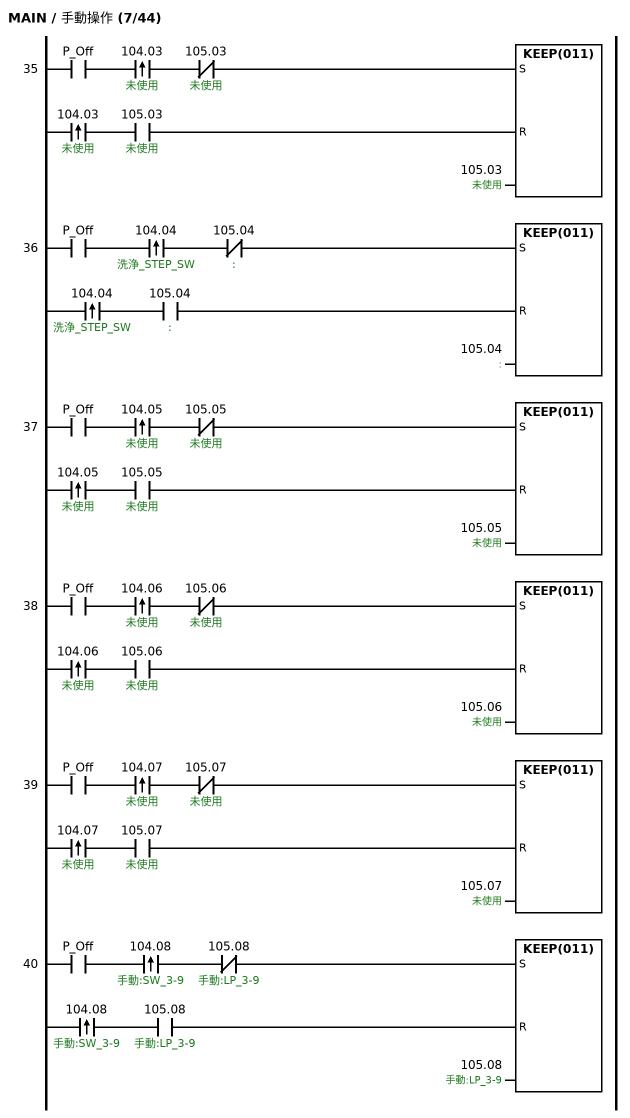
; rung 35
LD P_Off
@AND 104.03  ; 未使用
ANDNOT 105.03  ; 未使用
@LD 104.03  ; 未使用
AND 105.03  ; 未使用
KEEP(011) 105.03  ; 未使用
; rung 36
LD P_Off
@AND 104.04  ; 洗浄_STEP_SW
ANDNOT 105.04  ; :
@LD 104.04  ; 洗浄_STEP_SW
AND 105.04  ; :
KEEP(011) 105.04  ; :
; rung 37
LD P_Off
@AND 104.05  ; 未使用
ANDNOT 105.05  ; 未使用
@LD 104.05  ; 未使用
AND 105.05  ; 未使用
KEEP(011) 105.05  ; 未使用
; rung 38
LD P_Off
@AND 104.06  ; 未使用
ANDNOT 105.06  ; 未使用
@LD 104.06  ; 未使用
AND 105.06  ; 未使用
KEEP(011) 105.06  ; 未使用
; rung 39
LD P_Off
@AND 104.07  ; 未使用
ANDNOT 105.07  ; 未使用
@LD 104.07  ; 未使用
AND 105.07  ; 未使用
KEEP(011) 105.07  ; 未使用
; rung 40
LD P_Off
@AND 104.08  ; 手動:SW_3-9
ANDNOT 105.08  ; 手動:LP_3-9
@LD 104.08  ; 手動:SW_3-9
AND 105.08  ; 手動:LP_3-9
KEEP(011) 105.08  ; 手動:LP_3-9

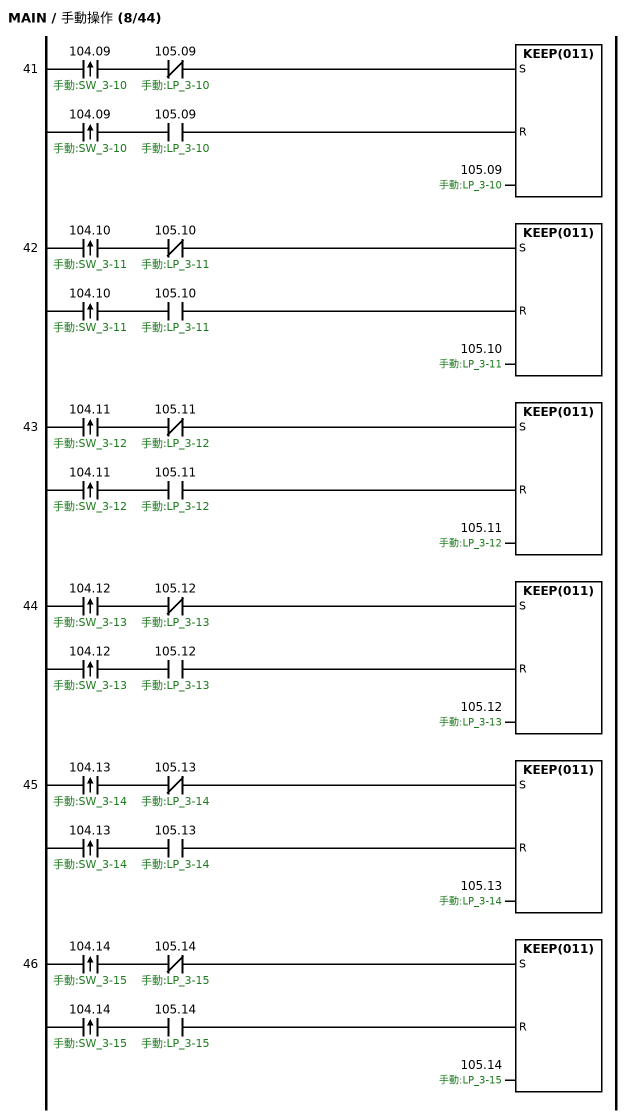
; rung 41
@LD 104.09  ; 手動:SW_3-10
ANDNOT 105.09  ; 手動:LP_3-10
@LD 104.09  ; 手動:SW_3-10
AND 105.09  ; 手動:LP_3-10
KEEP(011) 105.09  ; 手動:LP_3-10
; rung 42
@LD 104.10  ; 手動:SW_3-11
ANDNOT 105.10  ; 手動:LP_3-11
@LD 104.10  ; 手動:SW_3-11
AND 105.10  ; 手動:LP_3-11
KEEP(011) 105.10  ; 手動:LP_3-11
; rung 43
@LD 104.11  ; 手動:SW_3-12
ANDNOT 105.11  ; 手動:LP_3-12
@LD 104.11  ; 手動:SW_3-12
AND 105.11  ; 手動:LP_3-12
KEEP(011) 105.11  ; 手動:LP_3-12
; rung 44
@LD 104.12  ; 手動:SW_3-13
ANDNOT 105.12  ; 手動:LP_3-13
@LD 104.12  ; 手動:SW_3-13
AND 105.12  ; 手動:LP_3-13
KEEP(011) 105.12  ; 手動:LP_3-13
; rung 45
@LD 104.13  ; 手動:SW_3-14
ANDNOT 105.13  ; 手動:LP_3-14
@LD 104.13  ; 手動:SW_3-14
AND 105.13  ; 手動:LP_3-14
KEEP(011) 105.13  ; 手動:LP_3-14
; rung 46
@LD 104.14  ; 手動:SW_3-15
ANDNOT 105.14  ; 手動:LP_3-15
@LD 104.14  ; 手動:SW_3-15
AND 105.14  ; 手動:LP_3-15
KEEP(011) 105.14  ; 手動:LP_3-15

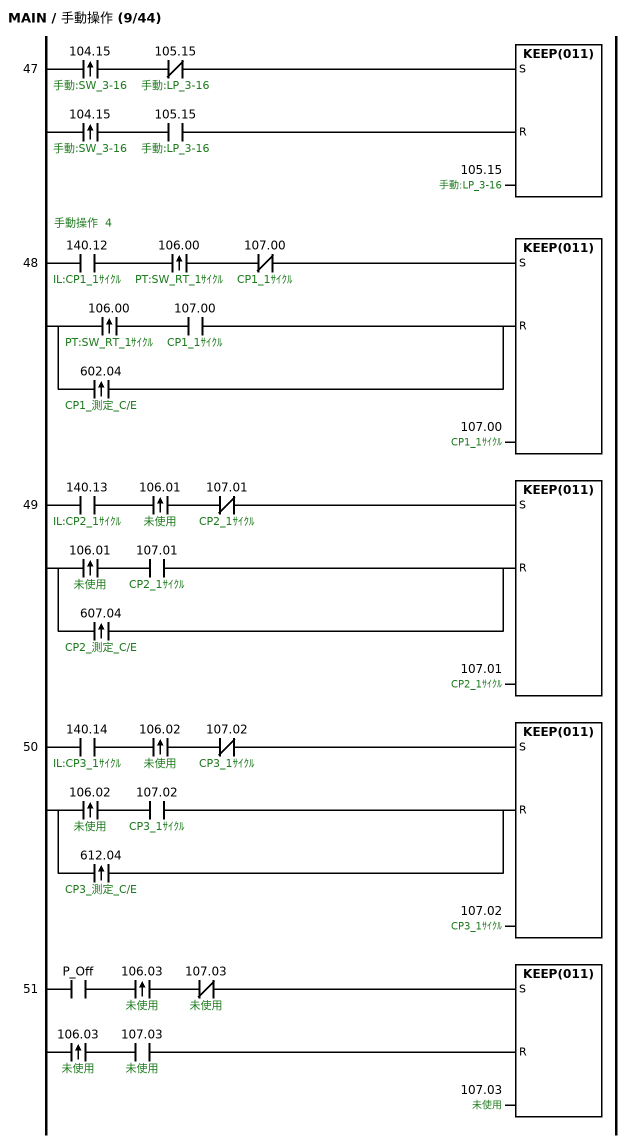
; rung 47
@LD 104.15  ; 手動:SW_3-16
ANDNOT 105.15  ; 手動:LP_3-16
@LD 104.15  ; 手動:SW_3-16
AND 105.15  ; 手動:LP_3-16
KEEP(011) 105.15  ; 手動:LP_3-16
; rung 48: 手動操作  4
LD 140.12  ; IL:CP1_1ｻｲｸﾙ
@AND 106.00  ; PT:SW_RT_1ｻｲｸﾙ
ANDNOT 107.00  ; CP1_1ｻｲｸﾙ
@LD 106.00  ; PT:SW_RT_1ｻｲｸﾙ
AND 107.00  ; CP1_1ｻｲｸﾙ
@OR 602.04  ; CP1_測定_C/E
KEEP(011) 107.00  ; CP1_1ｻｲｸﾙ
; rung 49
LD 140.13  ; IL:CP2_1ｻｲｸﾙ
@AND 106.01  ; 未使用
ANDNOT 107.01  ; CP2_1ｻｲｸﾙ
@LD 106.01  ; 未使用
AND 107.01  ; CP2_1ｻｲｸﾙ
@OR 607.04  ; CP2_測定_C/E
KEEP(011) 107.01  ; CP2_1ｻｲｸﾙ
; rung 50
LD 140.14  ; IL:CP3_1ｻｲｸﾙ
@AND 106.02  ; 未使用
ANDNOT 107.02  ; CP3_1ｻｲｸﾙ
@LD 106.02  ; 未使用
AND 107.02  ; CP3_1ｻｲｸﾙ
@OR 612.04  ; CP3_測定_C/E
KEEP(011) 107.02  ; CP3_1ｻｲｸﾙ
; rung 51
LD P_Off
@AND 106.03  ; 未使用
ANDNOT 107.03  ; 未使用
@LD 106.03  ; 未使用
AND 107.03  ; 未使用
KEEP(011) 107.03  ; 未使用

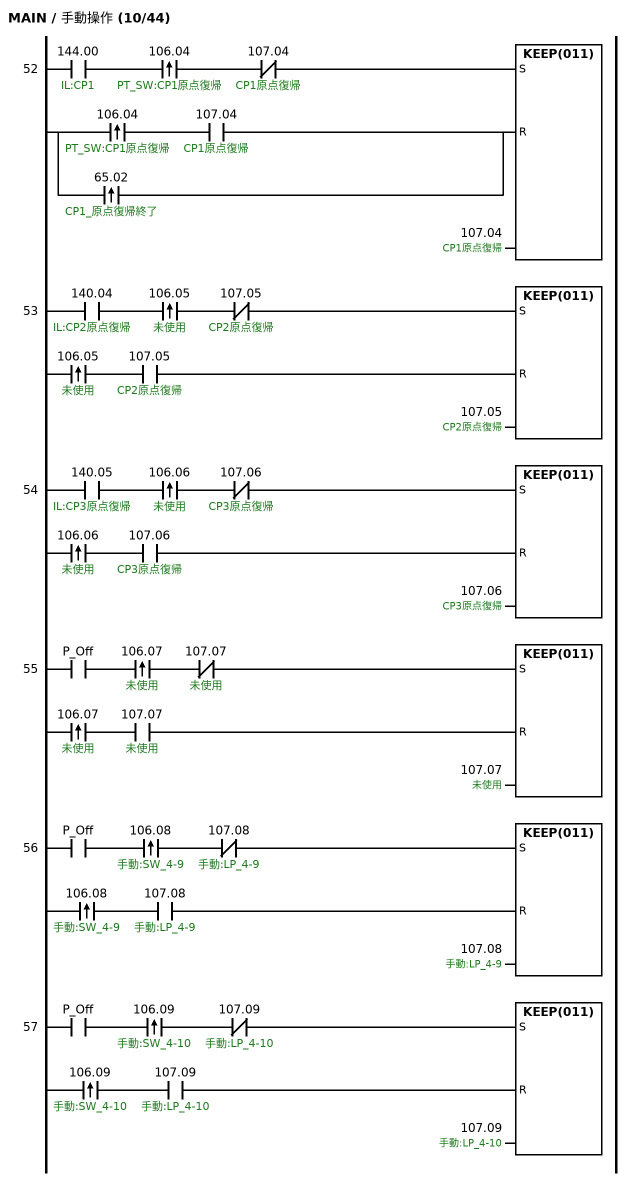
; rung 52
LD 144.00  ; IL:CP1
@AND 106.04  ; PT_SW:CP1原点復帰
ANDNOT 107.04  ; CP1原点復帰
@LD 106.04  ; PT_SW:CP1原点復帰
AND 107.04  ; CP1原点復帰
@OR 65.02  ; CP1_原点復帰終了
KEEP(011) 107.04  ; CP1原点復帰
; rung 53
LD 140.04  ; IL:CP2原点復帰
@AND 106.05  ; 未使用
ANDNOT 107.05  ; CP2原点復帰
@LD 106.05  ; 未使用
AND 107.05  ; CP2原点復帰
KEEP(011) 107.05  ; CP2原点復帰
; rung 54
LD 140.05  ; IL:CP3原点復帰
@AND 106.06  ; 未使用
ANDNOT 107.06  ; CP3原点復帰
@LD 106.06  ; 未使用
AND 107.06  ; CP3原点復帰
KEEP(011) 107.06  ; CP3原点復帰
; rung 55
LD P_Off
@AND 106.07  ; 未使用
ANDNOT 107.07  ; 未使用
@LD 106.07  ; 未使用
AND 107.07  ; 未使用
KEEP(011) 107.07  ; 未使用
; rung 56
LD P_Off
@AND 106.08  ; 手動:SW_4-9
ANDNOT 107.08  ; 手動:LP_4-9
@LD 106.08  ; 手動:SW_4-9
AND 107.08  ; 手動:LP_4-9
KEEP(011) 107.08  ; 手動:LP_4-9
; rung 57
LD P_Off
@AND 106.09  ; 手動:SW_4-10
ANDNOT 107.09  ; 手動:LP_4-10
@LD 106.09  ; 手動:SW_4-10
AND 107.09  ; 手動:LP_4-10
KEEP(011) 107.09  ; 手動:LP_4-10

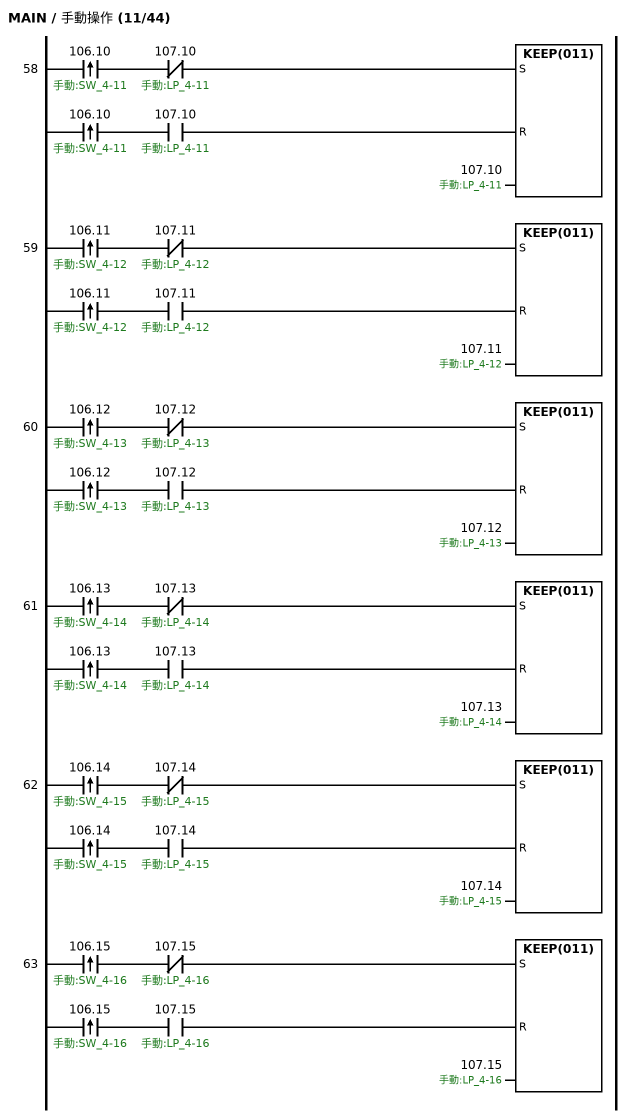
; rung 58
@LD 106.10  ; 手動:SW_4-11
ANDNOT 107.10  ; 手動:LP_4-11
@LD 106.10  ; 手動:SW_4-11
AND 107.10  ; 手動:LP_4-11
KEEP(011) 107.10  ; 手動:LP_4-11
; rung 59
@LD 106.11  ; 手動:SW_4-12
ANDNOT 107.11  ; 手動:LP_4-12
@LD 106.11  ; 手動:SW_4-12
AND 107.11  ; 手動:LP_4-12
KEEP(011) 107.11  ; 手動:LP_4-12
; rung 60
@LD 106.12  ; 手動:SW_4-13
ANDNOT 107.12  ; 手動:LP_4-13
@LD 106.12  ; 手動:SW_4-13
AND 107.12  ; 手動:LP_4-13
KEEP(011) 107.12  ; 手動:LP_4-13
; rung 61
@LD 106.13  ; 手動:SW_4-14
ANDNOT 107.13  ; 手動:LP_4-14
@LD 106.13  ; 手動:SW_4-14
AND 107.13  ; 手動:LP_4-14
KEEP(011) 107.13  ; 手動:LP_4-14
; rung 62
@LD 106.14  ; 手動:SW_4-15
ANDNOT 107.14  ; 手動:LP_4-15
@LD 106.14  ; 手動:SW_4-15
AND 107.14  ; 手動:LP_4-15
KEEP(011) 107.14  ; 手動:LP_4-15
; rung 63
@LD 106.15  ; 手動:SW_4-16
ANDNOT 107.15  ; 手動:LP_4-16
@LD 106.15  ; 手動:SW_4-16
AND 107.15  ; 手動:LP_4-16
KEEP(011) 107.15  ; 手動:LP_4-16

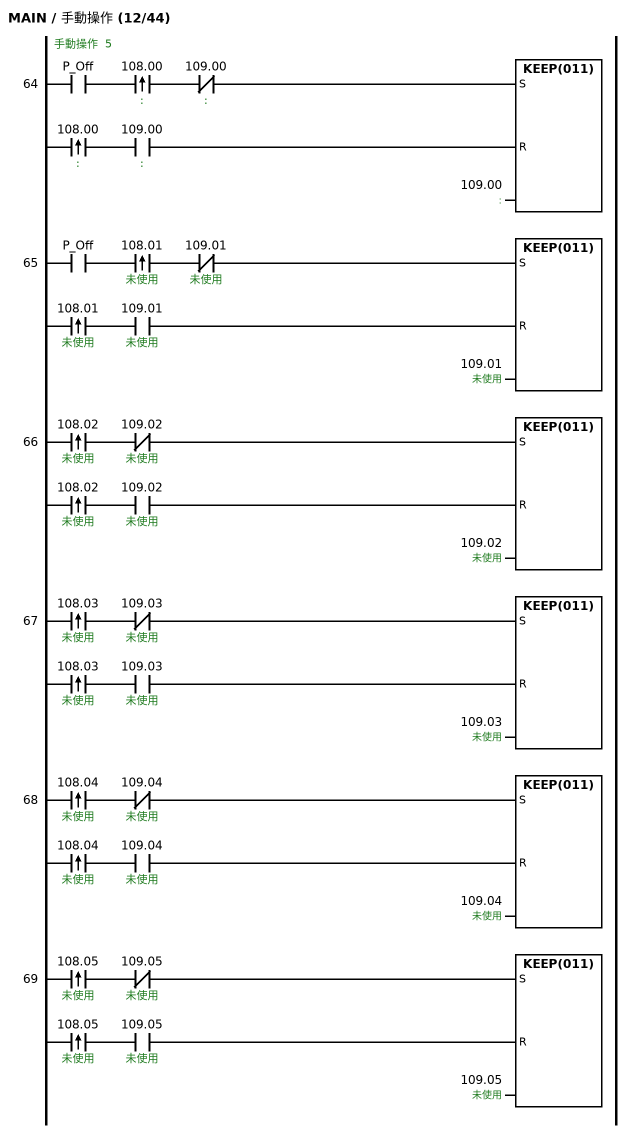
; rung 64: 手動操作  5
LD P_Off
@AND 108.00  ; :
ANDNOT 109.00  ; :
@LD 108.00  ; :
AND 109.00  ; :
KEEP(011) 109.00  ; :
; rung 65
LD P_Off
@AND 108.01  ; 未使用
ANDNOT 109.01  ; 未使用
@LD 108.01  ; 未使用
AND 109.01  ; 未使用
KEEP(011) 109.01  ; 未使用
; rung 66
@LD 108.02  ; 未使用
ANDNOT 109.02  ; 未使用
@LD 108.02  ; 未使用
AND 109.02  ; 未使用
KEEP(011) 109.02  ; 未使用
; rung 67
@LD 108.03  ; 未使用
ANDNOT 109.03  ; 未使用
@LD 108.03  ; 未使用
AND 109.03  ; 未使用
KEEP(011) 109.03  ; 未使用
; rung 68
@LD 108.04  ; 未使用
ANDNOT 109.04  ; 未使用
@LD 108.04  ; 未使用
AND 109.04  ; 未使用
KEEP(011) 109.04  ; 未使用
; rung 69
@LD 108.05  ; 未使用
ANDNOT 109.05  ; 未使用
@LD 108.05  ; 未使用
AND 109.05  ; 未使用
KEEP(011) 109.05  ; 未使用

